Fanuc KAREL source: kt00950.KL

PROGRAM KT00950
%STACKSIZE=65535
%PRIORITY=65535
%NOLOCKGROUP
VAR
ENTRY : INTEGER
PNAME : STRING[80]
VNAME : STRING[80]
STATUS : INTEGER
-- UNRESOLVED DECLARATIONS (source type spelling not recovered)
-- VALUE : ARRAY[4] OF TYPE_0x0017 (type_u16=0x2017)
BEGIN
ENTRY=0
PNAME=''
VNAME='VALUE'
-- UNRESOLVED_PC line 13 opcodes [27 22 22 2A 22 2A 22 22 AF] marker_code=43
END KT00950
